VAR_GLOBAL
	stMasterNetIdPhys AT %I* : T_AmsNetIdArr;	
	myInput AT %I*: BOOL;
	myOutput AT %Q*: BOOL;
END_VAR

(* stored: Version 1.1.0.1, ProductVersion 3.1.4024.3
   GVL GVL: Id {8169e3f9-6ee2-4370-afb9-efada7f02e64} *)
